// TIA Portal V18 export
FUNCTION "AIvars" : Void   // FC10014, LAD
{ S7_Optimized_Access := 'TRUE' }
VERSION : 0.1
// stored: AutoNumber false, IsIECCheckEnabled false, SetENOAutomatically false, UDAEnableTagReadback false
   VAR_INPUT
      rInput : Real;
      iFuncSystem : Byte;
      iFuncVar : Byte;
   END_VAR
BEGIN

REGION Network 1 (SCL)
   CASE #iFuncSystem OF
       0:  // Statement section case 2 to 4
           ;
       1..3:  // Statement section case 1
           CASE #iFuncVar OF
               0:  //
                   ;
               1:  //
                   "AHUAI".AI.rIAQ[#iFuncSystem] := #rInput;
               2:  // 
                   "AHUAI".AI.rBuildingdP[#iFuncSystem] := #rInput;
               3:  // 
                   "AHUAI".AI.rRoomAirTemp_PLC_AI[#iFuncSystem] := #rInput;
               4:  // 
                   "AHUAI".AI.rSupplyAirTemp[#iFuncSystem] := #rInput;
               5:  // 
                   "AHUAI".AI.rReturnAirTemp[#iFuncSystem] := #rInput;
               6:  // 
                   "AHUAI".AI.rFrostProtWaterTemp[#iFuncSystem] := #rInput;
               7:  // 
                   "AHUAI".AI.rFrostProtAirTemp[#iFuncSystem] := #rInput;
               8:  // 
                   "AHUAI".AI.rRoomAirRelHumi[#iFuncSystem] := #rInput;
               9:  // reserve
                   "AHUAI".AI.rReserve[#iFuncSystem] := #rInput;;
               10:  // 
                   "AHUAI".AI.rSAFilterdP[#iFuncSystem] := #rInput;
               11:
                   "AHUAI".AI.rSAFFlow[#iFuncSystem] := #rInput;
               12:
                   "AHUAI".AI.rRoomAirTemp_Actual[#iFuncSystem] := #rInput;
               13:
                   "AHUAI".AI.rRoomAirTemp_LoraAvg[#iFuncSystem] := #rInput;
               14:
                   "AHUAI".AI.rRoomAirTemp_MSensor[#iFuncSystem] := #rInput;
               ELSE
                   ;
           END_CASE;
       4..9:
           ;
       10:
           CASE #iFuncVar OF
               0:  // 
                   ;
               1:  // 
                   "HSsAI".AI.rHSBoilerRoomTemp := #rInput;
               2:  // 
                   "HSsAI".AI.rHSWaterPressure := #rInput;
               3:  // 
                   "HSsAI".AI.rHSSupplyMainfoldTemp := #rInput;
               4:  // 
                   "HSsAI".AI.rOutdoorTemp_PLC_AI := #rInput;
               5:    
                   "HCsAI".AI.rSupplyWaterTemp[1] := #rInput;
               6:  // 
                   "HCsAI".AI.rReturnWaterTemp[1] := #rInput;
               7:  // 
                   "HCsAI".AI.r3vwPosFbk[1] := #rInput;
               8:    
                   "HCsAI".AI.rSupplyWaterTemp[2] := #rInput;
               9:  // 
                   "HCsAI".AI.rReturnWaterTemp[2] := #rInput;
               10:  // 
                   "HCsAI".AI.r3vwPosFbk[2] := #rInput;
               ELSE
                   ;
           END_CASE;
       11..13:
           ;
       14:
           CASE #iFuncVar OF
               0:  // 
                   ;
               1:
                   "DHWAI".AI.r14200a := #rInput;
               2:  // 
                   "DHWAI".AI.r14201a := #rInput;
               ELSE
                   ;
           END_CASE;
       15..20:
           ;
       21: //Proxy Channels    
           CASE #iFuncVar OF
               0:  //
                   ;
               1..8:  //
                   "AHUProxyCH".Vars.rCHDrivenSignal[#iFuncVar] := #rInput;
               ELSE
                   ;
           END_CASE;
       22..99:
           ;
       100: //Diesel Line   
           CASE #iFuncVar OF
               0:  //
                   ;
               1:  //
                   "DLsAI".AI.rDayTankLevel[1] := #rInput;
               2:  //
                   "DLsAI".AI.rDayTankLevel[2] := #rInput;
               ELSE
                   ;
           END_CASE;
       ELSE  // Statement section ELSE
           ;
   END_CASE;
END_REGION
END_FUNCTION
